(*
SPDX-FileCopyrightText: © 2026 Oleksandr Tiutyk <trofimich@gmail.com>
SPDX-License-Identifier: MIT
License: https://opensource.org/license/mit
*)

(*!
<summary>Stores unique generic values with fixed or dynamic capacity.</summary>
<description>
CreateEnumerator allocates an independent cursor owned by its caller. The collection must remain alive while
that cursor is used. SetGeneric replaces a matching entry with the incoming descriptor. SetGeneric preserves
disposal responsibility when the same allocation is reused; transferred caller-side owning aliases must not be
released again. Lookup uses GENERIC_VALUE equality/hashing or the borrowed valueEqualityComparer supplied once
through FB_init. Pass zero explicitly to use default value equality and hashing. Empty values are supported
unless rejected by a validator. Raw queries create borrowed descriptors with an explicit object flag. Entries
and enumeration have no guaranteed order; positions are storage slots, not sorted ranks. Do not modify stored
descriptors through returned references. Try lookup/removal operations contain exceptions without rolling back
partial effects. Generic query arguments are borrowed by default. Explicitly requested release in Try
operations is attempted even after lookup failure; caller-side owning aliases are not reset. Borrowed
elements, including OBJECT instances, remain caller-owned and must stay alive while stored. Do not delete
owned payload through external aliases. Keep equality/hash-relevant data and comparer configuration stable:
remove before changing them, then insert again. Fields unrelated to active equality/hash may change. Callbacks
must not mutate elements or reenter collection mutation; explicit query release must not dispose of retained
storage. Default OBJECT equality/hashing uses Object.Equals/GetHashCode; Clone has its own identity. Discard
and populate the index again after equality-relevant address relocation before further lookup. Static index
storage adds 12 bytes per capacity slot and three pointers plus the comparer reference. Dynamic entries and
the 12-byte-per-slot index share one allocation; growth temporarily retains both old and new allocations.
Expected bucket lookup is constant time plus hashing/equality costs, worst case linear; compaction and
rebuilding after removal are linear in capacity and Length. The validator is borrowed for the collection
lifetime. No internal locking is implemented. Concurrent access involving mutation requires caller
coordination; this implementation does not provide a concurrent-container guarantee. Generic lookup with
requested query release also attempts cleanup on lookup failure before propagating the captured exception;
terminal OOM takes precedence.
Instances cannot be assigned by value: copying backing pointers or disposal responsibility would create
unsafe aliases. Interface references still borrow this instance; copying an interface does not clone storage.
</description>
*)

{attribute 'no_explicit_call' := 'do not call this function block directly'}
FUNCTION_BLOCK UniqueDataSet
VAR_GENERIC CONSTANT
	{attribute 'hide'}
	//! <summary>Inline capacity; zero selects dynamic backing storage.</summary>
	_StaticCapacity : TOF_Core.DINT_LENGTH := 0;
END_VAR
EXTENDS TOF_Core.Object IMPLEMENTS IUniqueDataSet
VAR_INPUT
	//! <summary>Number of slots added when dynamic storage is full; must be positive when growth is required.</summary>
	DefaultDynamicAllocationElementCount : BYTE := 10;
END_VAR
VAR_STAT
	//! <summary>Class name shared by all instances of this function block.</summary>
	{attribute 'hide'}
	_ClassName : STRING := __POUNAME();
END_VAR
VAR
	{attribute 'hide'}
	_ValueValidator : TOF_Core.IGenericValueValidator;
	{attribute 'hide'}
	_ValueEqualityComparer : TOF_Core.IEqualityComparer;

	{attribute 'hide'}
	_Array : POINTER TO TOF_Core.GENERIC_VALUE;
	{attribute 'hide'}
	_StaticArray : ARRAY [0.._StaticCapacity - 1] OF TOF_Core.GENERIC_VALUE;

	{attribute 'hide'}
	_Hashes : POINTER TO UDINT;
	{attribute 'hide'}
	_Buckets : POINTER TO DINT;
	{attribute 'hide'}
	_NextIndices : POINTER TO DINT;

	{attribute 'hide'}
	_StaticHashes : ARRAY [0.._StaticCapacity - 1] OF UDINT;
	{attribute 'hide'}
	_StaticBuckets : ARRAY [0.._StaticCapacity - 1] OF DINT;
	{attribute 'hide'}
	_StaticNextIndices : ARRAY [0.._StaticCapacity - 1] OF DINT;

	{attribute 'hide'}
	_DynamicCapacity : TOF_Core.DINT_LENGTH;
	{attribute 'hide'}
	_Length : TOF_Core.DINT_LENGTH;
END_VAR

(*!
<summary>Grows the combined entry and hash-index buffer before accepting incoming ownership.</summary>
<description>
Static collections return without allocation. A positive increment must fit DINT capacity and the UDINT
allocation-byte limit, including 12 index bytes per slot. One allocation contains entries, cached hashes,
bucket heads and links. Allocation failure preserves the old buffer, index, capacity and payload ownership and
sets terminal allocation state. Existing descriptors and hashes are copied; rebuilding links invokes no
equality/hash callbacks. Descendants cannot override this storage operation; capacity, indexing and disposal
remain governed by this collection implementation.
</description>
*)
METHOD PROTECTED FINAL AllocateMemory
VAR_INPUT
	elementCount : TOF_Core.DINT_LENGTH;
END_VAR
VAR CONSTANT
	//! <summary>Bytes per capacity slot, including descriptor storage and any hash-index arrays.</summary>
	ENTRY_ALLOCATION_SIZE : ULINT := XSIZEOF(TOF_Core.GENERIC_VALUE) + XSIZEOF(UDINT) + 2 * XSIZEOF(DINT);
END_VAR
VAR
	newMemory : POINTER TO BYTE;
	newHashes : POINTER TO UDINT;
	newCapacity : ULINT;

END_VAR
IF NOT Dynamic THEN
	RETURN;
END_IF

IF elementCount <= TOF_Core.SignedInt32.ZERO THEN
	TOF_Core.Exceptions.ThrowArgumentOutOfRange(
		sourceNamespaceName := NamespaceName,
		sourceClassName := ClassName,
		sourcePOUName := __POUNAME(),
		sourcePosition := __POSITION(),
		argumentName := 'elementCount',
		argumentValue := elementCount
	);
END_IF

newCapacity := TO_ULINT(_DynamicCapacity) + TO_ULINT(elementCount);

IF newCapacity > TO_ULINT(TOF_Core.SignedInt32.MAX_VALUE)
	OR_ELSE newCapacity > TO_ULINT(TOF_Core.UnsignedInt32.MAX_VALUE) / ENTRY_ALLOCATION_SIZE
THEN
	TOF_Core.Exceptions.ThrowArgumentOutOfRange(
		sourceNamespaceName := NamespaceName,
		sourceClassName := ClassName,
		sourcePOUName := __POUNAME(),
		sourcePosition := __POSITION(),
		argumentName := 'capacity',
		argumentValue := newCapacity
	);
END_IF

newMemory := __NEW(BYTE, TO_UDINT(ENTRY_ALLOCATION_SIZE * newCapacity));

IF newMemory = 0 THEN
	TOF_Core.DynamicMemoryManager.RaiseAllocationFailure();
END_IF

newHashes := newMemory + TO_UDINT(XSIZEOF(TOF_Core.GENERIC_VALUE) * newCapacity);

IF _Length > TOF_Core.SignedInt32.ZERO THEN
	Tc2_System.MEMCPY(
		destAddr := newMemory,
		srcAddr := _Array,
		n := TO_UDINT(XSIZEOF(TOF_Core.GENERIC_VALUE) * TO_ULINT(_Length))
	);
	Tc2_System.MEMCPY(destAddr := newHashes, srcAddr := _Hashes, n := TO_UDINT(XSIZEOF(UDINT) * TO_ULINT(_Length)));
END_IF

IF _Array <> 0 THEN
	__DELETE(_Array);
END_IF

_Array := newMemory;
_Hashes := newHashes;
_Buckets := newMemory + TO_UDINT((XSIZEOF(TOF_Core.GENERIC_VALUE) + XSIZEOF(UDINT)) * newCapacity);
_NextIndices := newMemory + TO_UDINT((XSIZEOF(TOF_Core.GENERIC_VALUE) + XSIZEOF(UDINT) + XSIZEOF(DINT)) * newCapacity);
_DynamicCapacity := TO_DINT(newCapacity);

rebuildIndex();
END_METHOD

(*!
<summary>Reports the currently allocated number of slots.</summary>
<description>
Units are bytes for ByteList and entries for other collections. Static capacity is fixed; dynamic capacity can
change on growth or clearing. This is not a guarantee that the next allocation succeeds.
</description>
*)
{attribute 'monitoring' := 'call'}
PROPERTY FINAL Capacity : TOF_Core.DINT_LENGTH
GET
Capacity := SEL(_StaticCapacity = 0, _StaticCapacity, _DynamicCapacity);
END_GET
END_PROPERTY

(*!
<summary>Borrows the concrete collection class name without transferring storage ownership.</summary>
*)
{attribute 'monitoring' := 'call'}
PROPERTY ClassName : REFERENCE TO STRING
GET
ClassName REF= _ClassName;
END_GET
END_PROPERTY

(*!
<summary>Removes all entries and releases dynamic entry and index storage.</summary>
<description>
Owned payload cleanup is best effort. The collection is marked empty before disposal; cleanup callbacks must
not reenter mutation. Static capacity and the lifetime comparer/validators are retained. Dynamic capacity
becomes zero. Uses no allocation or equality/hash callbacks and leaves static buckets empty for reuse.
Descendants cannot override this storage operation; capacity, indexing and disposal remain governed by this
collection implementation.
</description>
*)
METHOD FINAL Clear : IUniqueDataSet
VAR
	index : DINT;
	entryCount : DINT;
END_VAR
Clear := THIS^;
entryCount := _Length;
_Length := 0;

FOR index := 0 TO entryCount - 1 DO
	_Array[index].Release();
END_FOR

IF Dynamic THEN
	IF _Array <> 0 THEN
		__DELETE(_Array);
	END_IF

	_Array := 0;
	_Hashes := 0;
	_Buckets := 0;
	_NextIndices := 0;
	_DynamicCapacity := 0;
ELSE
	rebuildIndex();
END_IF
END_METHOD

(*!
<summary>Reports whether a matching raw query exists.</summary>
<description>
The raw ANY argument is borrowed without cloning or ownership transfer. isObject = TRUE requires a live Object
function-block instance, not a pointer or interface variable. FALSE uses ordinary runtime type mapping. The
caller keeps the query storage alive for the call. Descendants cannot override this storage operation;
capacity, indexing and disposal remain governed by this collection implementation.
</description>
*)
//!<param name="isObject">Explicitly interprets the raw argument as a live Object instance.</param>
METHOD FINAL Contains : BOOL
VAR_INPUT
	value : ANY;
	isObject : BOOL := FALSE;
END_VAR
VAR
	genericValue : TOF_Core.GENERIC_VALUE;
END_VAR

genericValue := TOF_Core.GenericValueFactory.FromAnyType(
		value := value,
		isObject := isObject,
		memoryManagementBehavior := TOF_Core.GENERIC_MEMORY_MANAGEMENT_BEHAVIOR.STORE_ORIGINAL_REFERENCE_AND_NOT_OWNS_MEMORY
	);

Contains := FindIndex(value := genericValue);
END_METHOD

(*!
<summary>Reports whether a matching entry exists for a borrowed generic query.</summary>
<description>
The query is borrowed by default. Explicit release requests disposal of owned query storage after lookup
completes, including a missing result. Requested release is attempted after both successful lookup and lookup
failure. Before cleanup, the original framework exception is retained and a borrowed static system exception
is cloned to preserve its code, catch point and timestamps across cleanup callbacks. The captured exception is
then propagated through ExceptionManager.Throw in the current cyclic task; native errors use the framework
SystemException representation. If capturing the system exception fails with terminal OOM, query cleanup is
still attempted and terminal OOM takes precedence. Terminal allocation state is never cleared. Release is best
effort and does not prove successful deallocation. Cleanup callbacks must not reenter collection mutation.
Release resets only the local descriptor copy; the caller must have disposal rights and must not reuse or
release owning aliases afterwards. Borrowed payload is not freed. Descendants cannot override this storage
operation; capacity, indexing and disposal remain governed by this collection implementation.
</description>
*)
METHOD FINAL ContainsGeneric : BOOL
VAR_INPUT
	value : TOF_Core.GENERIC_VALUE;
	releaseValue : BOOL := FALSE;
END_VAR
VAR
	exceptionCode : __SYSTEM.ExceptionCode;
	caughtException : TOF_Core.IException;
END_VAR
__TRY
	ContainsGeneric := FindIndex(value := value);
__CATCH(exceptionCode)
	caughtException := TOF_Core.ExceptionManager.GetLastException(
		exceptionCode := exceptionCode,
		catchPointNamespaceName := NamespaceName,
		catchPointPOUName := __POUNAME(),
		catchPointPosition := __POSITION()
	);
__ENDTRY

IF releaseValue THEN
	IF caughtException <> 0 AND_THEN NOT caughtException.IsDynamicInstance THEN
		__TRY
			TOF_Core.DynamicMemoryManager.RaiseIfAllocationFailed();
			__QUERYINTERFACE(caughtException.Clone(), caughtException);
		__CATCH(exceptionCode)
			value.Release();

			TOF_Core.ExceptionManager.ReThrowLastException(
				exceptionCode := exceptionCode,
				catchPointNamespaceName := NamespaceName,
				catchPointPOUName := __POUNAME(),
				catchPointPosition := __POSITION()
			);
		__ENDTRY
	END_IF

	value.Release();
END_IF

IF caughtException <> 0 THEN
	TOF_Core.ExceptionManager.Throw(exception := caughtException);
END_IF
END_METHOD

(*!
<summary>Creates an independent enumerator owned by the caller.</summary>
<description>
The caller must explicitly release the enumerator and keep this collection alive while using it. Allocation
failure invokes DynamicMemoryManager.RaiseAllocationFailure without a heap exception; it is terminal and is
not returned as a recoverable null result.
</description>
*)
METHOD CreateEnumerator : TOF_Core.IEnumerator
VAR
	enumerator : POINTER TO UniqueDataSetEnumerator;
END_VAR
enumerator := __NEW(UniqueDataSetEnumerator(uniqueSet := THIS^));

IF enumerator = 0 THEN
	TOF_Core.DynamicMemoryManager.RaiseAllocationFailure();
END_IF

CreateEnumerator := enumerator^;
END_METHOD

(*!
<summary>Reports whether storage can grow dynamically.</summary>
<description>
Static capacity zero selects dynamic storage. Dynamic collections can still fail to allocate.
</description>
*)
{attribute 'monitoring' := 'call'}
PROPERTY FINAL Dynamic : BOOL
GET
Dynamic := _StaticCapacity = 0;
END_GET
END_PROPERTY

(*!
<summary>Reports whether the collection has no entries.</summary>
<description>
Reflects Length; not a check of payload lifetime or memory health.
</description>
*)
{attribute 'monitoring' := 'call'}
PROPERTY FINAL Empty : BOOL
GET
Empty := _Length <= 0;
END_GET
END_PROPERTY

(*!
<summary>Releases collection payload and dynamic entry/index storage during destruction.</summary>
<description>
Calls the non-allocating Clear path without invoking equality/hash callbacks. Owned payload release is best
effort and cannot guarantee successful deallocation; cleanup callbacks must not throw or reenter mutation.
</description>
*)

METHOD FB_exit : BOOL
VAR_INPUT
	bInCopyCode : BOOL;
END_VAR
Clear();
END_METHOD

(*!
<summary>Binds the validator, the lifetime equality strategy and static storage.</summary>
<description>
The value comparer is borrowed for the entire collection lifetime. Supply it explicitly; zero selects
GENERIC_VALUE default equality and hashing. Keep it alive and its equality-relevant configuration stable.
There is no subsequent comparer replacement. Initialization binds existing storage without allocating or
calling validators, comparers or other throwing paths.
</description>
*)


//!<param name="valueEqualityComparer">
//! Borrowed value equality and hash strategy; pass zero explicitly for the GENERIC_VALUE defaults.
//! </param>
METHOD FB_init : BOOL
VAR_INPUT
	bInitRetains : BOOL; // TRUE: the retain variables are initialized (reset warm / reset cold)
	bInCopyCode : BOOL; // TRUE: the instance will be copied to the copy code afterward (online change)

	valueValidator : TOF_Core.IGenericValueValidator;
	valueEqualityComparer : TOF_Core.IEqualityComparer;
END_VAR
_ValueValidator := valueValidator;
_ValueEqualityComparer := valueEqualityComparer;

IF NOT Dynamic THEN
	_Array := ADR(_StaticArray);
	_Hashes := ADR(_StaticHashes);
	_Buckets := ADR(_StaticBuckets);
	_NextIndices := ADR(_StaticNextIndices);
END_IF
END_METHOD

(*!
<summary>Finds an equal value through its hash bucket.</summary>
<description>
Borrows the descriptor and payload without changing ownership. The configured equality strategy computes the
query hash once; equal hash codes are resolved with Equals. Callback exceptions propagate before mutation. On
a miss supposedIndex is the append position. hashCode is valid after a completed lookup, including a miss. No
ordering or sorted rank is provided. Bucket heads and links encode entry index plus one; zero ends a chain.
Descendants cannot override this storage operation; capacity, indexing and disposal remain governed by this
collection implementation.
</description>
*)
METHOD PROTECTED FINAL FindIndex : BOOL
VAR_INPUT
	value : TOF_Core.GENERIC_VALUE;
END_VAR
VAR_OUTPUT
	supposedIndex : DINT;
	hashCode : UDINT;
END_VAR
VAR
	entryLink : DINT;
	entryIndex : DINT;
END_VAR
FindIndex := FALSE;
supposedIndex := _Length;
hashCode := value.GetHashCode(comparer := _ValueEqualityComparer);

IF _Length = TOF_Core.SignedInt32.ZERO THEN
	RETURN;
END_IF

entryLink := _Buckets[TO_DINT(hashCode MOD TO_UDINT(Capacity))];

WHILE entryLink <> TOF_Core.SignedInt32.ZERO DO
	entryIndex := entryLink - 1;

	IF _Hashes[entryIndex] = hashCode
		AND_THEN _Array[entryIndex].Equals(otherValue := value, comparer := _ValueEqualityComparer)
	THEN
		supposedIndex := entryIndex;
		FindIndex := TRUE;
		RETURN;
	END_IF

	entryLink := _NextIndices[entryIndex];
END_WHILE
END_METHOD

(*!
<summary>Reports whether fixed-capacity storage has no free slot.</summary>
<description>
Dynamic collections report FALSE even when Length equals Capacity. This does not guarantee available heap
memory.
</description>
*)
{attribute 'monitoring' := 'call'}
PROPERTY FINAL Full : BOOL
GET
Full := _StaticCapacity <> 0 AND_THEN _Length >= _StaticCapacity;
END_GET
END_PROPERTY

(*!
<summary>Borrows the entry at a current storage position.</summary>
<description>
The index must be within Length and is not a sorted rank; otherwise an exception is raised. The returned
descriptor reference and payload remain collection-owned or borrowed from their original owner. Do not mutate
the descriptor or dispose of its payload through this view. Mutation or destruction may invalidate the
reference. Descendants cannot override this storage operation; capacity, indexing and disposal remain governed
by this collection implementation.
</description>
*)
METHOD FINAL GetByIndex : REFERENCE TO TOF_Core.GENERIC_VALUE
VAR_INPUT
	index : DINT;
END_VAR
IF index < 0 OR_ELSE index >= _Length THEN
	TOF_Core.Exceptions.ThrowArgumentOutOfRange(
		sourceNamespaceName := NamespaceName,
		sourceClassName := ClassName,
		sourcePOUName := __POUNAME(),
		sourcePosition := __POSITION(),
		argumentName := 'index',
		argumentValue := index
	);
END_IF

GetByIndex REF= _Array[index];
END_METHOD

(*!
<summary>Returns the matching entry position, or a negative value when absent.</summary>
<description>
The query is borrowed by default. Explicit release requests disposal of owned query storage after lookup
completes, including a missing result. Requested release is attempted after both successful lookup and lookup
failure. Before cleanup, the original framework exception is retained and a borrowed static system exception
is cloned to preserve its code, catch point and timestamps across cleanup callbacks. The captured exception is
then propagated through ExceptionManager.Throw in the current cyclic task; native errors use the framework
SystemException representation. If capturing the system exception fails with terminal OOM, query cleanup is
still attempted and terminal OOM takes precedence. Terminal allocation state is never cleared. Release is best
effort and does not prove successful deallocation. Cleanup callbacks must not reenter collection mutation.
Release resets only the local descriptor copy; the caller must have disposal rights and must not reuse or
release owning aliases afterwards. Borrowed payload is not freed. The position is a current storage slot with
no sorted-rank guarantee; mutation may invalidate it. Descendants cannot override this storage operation;
capacity, indexing and disposal remain governed by this collection implementation.
</description>
*)
METHOD FINAL GetGenericValuePosition : DINT
VAR_INPUT
	value : TOF_Core.GENERIC_VALUE;
	releaseValue : BOOL := FALSE;
END_VAR
VAR
	exceptionCode : __SYSTEM.ExceptionCode;
	caughtException : TOF_Core.IException;
END_VAR
__TRY
	IF NOT FindIndex(value := value, supposedIndex => GetGenericValuePosition) THEN
		GetGenericValuePosition := -1;
	END_IF
__CATCH(exceptionCode)
	caughtException := TOF_Core.ExceptionManager.GetLastException(
		exceptionCode := exceptionCode,
		catchPointNamespaceName := NamespaceName,
		catchPointPOUName := __POUNAME(),
		catchPointPosition := __POSITION()
	);
__ENDTRY

IF releaseValue THEN
	IF caughtException <> 0 AND_THEN NOT caughtException.IsDynamicInstance THEN
		__TRY
			TOF_Core.DynamicMemoryManager.RaiseIfAllocationFailed();
			__QUERYINTERFACE(caughtException.Clone(), caughtException);
		__CATCH(exceptionCode)
			value.Release();

			TOF_Core.ExceptionManager.ReThrowLastException(
				exceptionCode := exceptionCode,
				catchPointNamespaceName := NamespaceName,
				catchPointPOUName := __POUNAME(),
				catchPointPosition := __POSITION()
			);
		__ENDTRY
	END_IF

	value.Release();
END_IF

IF caughtException <> 0 THEN
	TOF_Core.ExceptionManager.Throw(exception := caughtException);
END_IF
END_METHOD

(*!
<summary>Returns the matching storage position, or a negative value when absent.</summary>
<description>
The raw ANY argument is borrowed without cloning or ownership transfer. isObject = TRUE requires a live Object
function-block instance, not a pointer or interface variable. FALSE uses ordinary runtime type mapping. The
caller keeps the query storage alive for the call. The position is a current storage slot with no sorted-rank
guarantee; mutation may invalidate it. Descendants cannot override this storage operation; capacity, indexing
and disposal remain governed by this collection implementation.
</description>
*)
//!<param name="isObject">Explicitly interprets the raw argument as a live Object instance.</param>
METHOD FINAL GetValuePosition : DINT
VAR_INPUT
	value : ANY;
	isObject : BOOL := FALSE;
END_VAR
VAR
	genericValue : TOF_Core.GENERIC_VALUE;
END_VAR

genericValue := TOF_Core.GenericValueFactory.FromAnyType(
		value := value,
		isObject := isObject,
		memoryManagementBehavior := TOF_Core.GENERIC_MEMORY_MANAGEMENT_BEHAVIOR.STORE_ORIGINAL_REFERENCE_AND_NOT_OWNS_MEMORY
	);

IF NOT FindIndex(value := genericValue, supposedIndex => GetValuePosition) THEN
	GetValuePosition := -1;
END_IF
END_METHOD

(*!
<summary>Reports the number of stored entries.</summary>
<description>
Units are bytes for ByteList and entries for other collections. Existing positions range from zero through
Length minus one.
</description>
*)
{attribute 'monitoring' := 'call'}
PROPERTY FINAL Length : TOF_Core.DINT_LENGTH
GET
Length := _Length;
END_GET
END_PROPERTY

(*!
<summary>Provides the library namespace for diagnostics.</summary>
<description>
Borrowed read-only reference to compiler-initialized metadata; no ownership transfer.
</description>
*)
{attribute 'monitoring' := 'call'}
PROPERTY NamespaceName : REFERENCE TO STRING
GET
NamespaceName REF= CurrentNamespace.Name;
END_GET
END_PROPERTY

(*!
<summary>Rebuilds bucket chains from cached hashes after entry relocation or capacity changes.</summary>
<description>
Requires bound index storage for positive capacity and valid hashes for every live entry. Does not allocate,
access payload or invoke callbacks. This only rebuilds links; it does not recompute hashes after
equality-relevant payload or address changes.
</description>
*)
METHOD PRIVATE rebuildIndex
VAR
	index : DINT;
	bucketIndex : DINT;
END_VAR
IF Capacity = TOF_Core.SignedInt32.ZERO THEN
	RETURN;
END_IF

Tc2_System.MEMSET(destAddr := _Buckets, fillByte := 0, n := TO_UDINT(XSIZEOF(DINT) * TO_ULINT(Capacity)));

FOR index := 0 TO _Length - 1 DO
	bucketIndex := TO_DINT(_Hashes[index] MOD TO_UDINT(Capacity));
	_NextIndices[index] := _Buckets[bucketIndex];
	_Buckets[bucketIndex] := index + 1;
END_FOR
END_METHOD

(*!
<summary>Removes the entry at a current storage position.</summary>
<description>
The index must be within Length and is not a sorted rank. Entries after the removed slot are compacted and
bucket links rebuilt from cached hashes before owned payload cleanup. Index compaction and rebuilding invoke
no equality/hash callbacks and allocate no storage. Invalid indices raise an exception. Positions and borrowed
entry references may be invalidated. Payload disposal is best effort through GENERIC_VALUE.Release.
Descendants cannot override this storage operation; capacity, indexing and disposal remain governed by this
collection implementation.
</description>
*)
METHOD FINAL RemoveAt : IUniqueDataSet
VAR_INPUT
	index : DINT;
END_VAR
VAR
	removedValue : TOF_Core.GENERIC_VALUE;
END_VAR
IF index < TOF_Core.SignedInt32.ZERO OR_ELSE index >= _Length THEN
	TOF_Core.Exceptions.ThrowArgumentOutOfRange(
		sourceNamespaceName := NamespaceName,
		sourceClassName := ClassName,
		sourcePOUName := __POUNAME(),
		sourcePosition := __POSITION(),
		argumentName := 'index',
		argumentValue := index
	);
END_IF

RemoveAt := THIS^;
removedValue := _Array[index];

IF index < _Length - 1 THEN
	Tc2_System.MEMMOVE(
		destAddr := ADR(_Array[index]),
		srcAddr := ADR(_Array[index + 1]),
		n := TO_UDINT(XSIZEOF(TOF_Core.GENERIC_VALUE) * TO_ULINT(_Length - index - 1))
	);
	Tc2_System.MEMMOVE(
		destAddr := ADR(_Hashes[index]),
		srcAddr := ADR(_Hashes[index + 1]),
		n := TO_UDINT(XSIZEOF(UDINT) * TO_ULINT(_Length - index - 1))
	);
END_IF

_Array[_Length - 1].Reset();
_Length := _Length - 1;
rebuildIndex();

removedValue.Release();
END_METHOD

(*!
<summary>Reports the size of this function-block instance.</summary>
<description>
Measured in bytes; includes inline storage but excludes separately allocated buffers, payload and enumerators.
</description>
*)
{attribute 'monitoring' := 'call'}
PROPERTY SelfSize : ULINT
GET
SelfSize := XSIZEOF(THIS^);
END_GET
END_PROPERTY

(*!
<summary>Copies a value and stores it through SetGeneric.</summary>
<description>
Borrows the original during the call. isObject = TRUE requires a live Object FB instance implementing
ICloneable; other data is copied as bytes without recursively cloning references. A prepared copy is released
if insertion fails before acceptance; exceptions propagate. Engine-managed exception objects are unsupported.
Any index output is meaningful only on success. Descendants cannot override this storage operation; capacity,
indexing and disposal remain governed by this collection implementation.
The original failure is captured before cleanup so nested cleanup handling cannot replace its payload.
A static native wrapper is cloned before cleanup; failure to capture still attempts prepared-copy disposal.
Terminal allocation failure takes precedence and no exception clone is allocated after its latch is set.
</description>
*)
METHOD FINAL SetCopy : IUniqueDataSet
VAR_INPUT
	value : ANY;
	isObject : BOOL := FALSE;
END_VAR
VAR_OUTPUT
	index : DINT;
END_VAR
VAR
	exceptionCode : __SYSTEM.ExceptionCode;
	caughtException : TOF_Core.IException;
	genericValue : TOF_Core.GENERIC_VALUE;
END_VAR

genericValue := TOF_Core.GenericValueFactory.FromAnyType(
		value := value,
		isObject := isObject,
		memoryManagementBehavior := TOF_Core.GENERIC_MEMORY_MANAGEMENT_BEHAVIOR.CLONE_ORIGINAL_VALUE_AND_OWNS_MEMORY
	);

__TRY
	SetCopy := SetGeneric(value := genericValue, index => index);
__CATCH(exceptionCode)
	caughtException := TOF_Core.ExceptionManager.GetLastException(
		exceptionCode := exceptionCode,
		catchPointNamespaceName := NamespaceName,
		catchPointPOUName := __POUNAME(),
		catchPointPosition := __POSITION()
	);
__ENDTRY

IF caughtException <> 0 THEN
	__TRY
		TOF_Core.DynamicMemoryManager.RaiseIfAllocationFailed();

		IF NOT caughtException.IsDynamicInstance THEN
			__QUERYINTERFACE(caughtException.Clone(), caughtException);
		END_IF
	__CATCH(exceptionCode)
		genericValue.Release();

		TOF_Core.ExceptionManager.ReThrowLastException(
			exceptionCode := exceptionCode,
			catchPointNamespaceName := NamespaceName,
			catchPointPOUName := __POUNAME(),
			catchPointPosition := __POSITION()
		);
	__ENDTRY

	genericValue.Release();

	TOF_Core.ExceptionManager.Throw(exception := caughtException);
END_IF
END_METHOD

(*!
<summary>Inserts a value or replaces the matching entry with the incoming descriptor.</summary>
<description>
Uses the lifetime equality/hash strategy, with no ordering guarantee. Empty descriptors are permitted unless
rejected by a validator. A successful call accepts incoming owned storage; borrowed payload must remain alive
while stored. Validation, lookup and growth precede acceptance; failure before acceptance leaves ownership
with the caller. A displaced owned allocation is released after replacement. Reusing the same allocation does
not release it and preserves existing ownership or accepts incoming ownership, without implicitly returning
ownership to the caller. Caller-side descriptor copies are not reset; transferred owning aliases must not be
released or reused as owners. Aliases must have compatible disposal semantics; overlapping owned ranges and
ownership already held by another entry or owner are not supported. Callbacks must not mutate or reenter this
collection. Cleanup through GENERIC_VALUE.Release is best effort and does not guarantee deallocation. The
index output is valid only on success. Descendants cannot override this storage operation; capacity, indexing
and disposal remain governed by this collection implementation.
</description>
*)
//!<param name="value">Incoming descriptor; owned storage is transferred on success.</param>
METHOD FINAL SetGeneric : IUniqueDataSet
VAR_INPUT
	value : TOF_Core.GENERIC_VALUE;
END_VAR
VAR_OUTPUT
	index : DINT;
END_VAR
VAR

	supposedIndex : DINT;
	hashCode : UDINT;
	bucketIndex : DINT;

	displacedValue : TOF_Core.GENERIC_VALUE;
END_VAR
IF _ValueValidator <> 0 THEN
	_ValueValidator.Validate(validatedObjectName := GetName(), valueToValidate := value);
END_IF

SetGeneric := THIS^;

IF FindIndex(value := value, supposedIndex => supposedIndex, hashCode => hashCode) THEN
	displacedValue := _Array[supposedIndex];

	IF displacedValue.Address = value.Address THEN
		IF displacedValue.IsMemoryOwner AND_THEN NOT value.IsMemoryOwner THEN
			value := TOF_Core.GenericValueFactory.FromParts(
				genericTypeClass := value.TypeClass,
				address := value.Address,
				size := value.Size,
				memoryManagementBehavior := TOF_Core.GENERIC_MEMORY_MANAGEMENT_BEHAVIOR.STORE_ORIGINAL_REFERENCE_AND_OWNS_MEMORY
			);
		END_IF

		displacedValue.Reset();
	END_IF
ELSE
	IF _Length >= Capacity THEN
		IF Dynamic THEN
			AllocateMemory(elementCount := DefaultDynamicAllocationElementCount);
		ELSE
			TOF_Core.Exceptions.ThrowStaticCollectionFull(
				sourceNamespaceName := NamespaceName,
				sourceClassName := ClassName,
				sourcePOUName := __POUNAME(),
				sourcePosition := __POSITION(),
				collectionName := GetName(),
				capacity := TO_UDINT(Capacity)
			);
		END_IF
	END_IF
END_IF

_Array[supposedIndex] := value;

IF supposedIndex = _Length THEN
	_Hashes[supposedIndex] := hashCode;
	bucketIndex := TO_DINT(hashCode MOD TO_UDINT(Capacity));
	_NextIndices[supposedIndex] := _Buckets[bucketIndex];
	_Buckets[bucketIndex] := supposedIndex + 1;
	_Length := _Length + 1;
END_IF

displacedValue.Release();

index := supposedIndex;
END_METHOD

(*!
<summary>Attempts to remove a matching entry.</summary>
<description>
Returns the collection for chaining. removed is TRUE only after the matching entry has been removed; FALSE
means no completed removal was reported. Removal is not transactional and does not prove successful
destruction of an owned payload. Catches exceptions without propagating them or clearing terminal allocation
state. Partial changes are not rolled back. The raw ANY argument is borrowed without cloning or ownership
transfer. isObject = TRUE requires a live Object function-block instance, not a pointer or interface variable.
FALSE uses ordinary runtime type mapping. The caller keeps the query storage alive for the call. Descendants
cannot override this storage operation; capacity, indexing and disposal remain governed by this collection
implementation.
After nested calls and requested cleanup, a fatal allocation state forces the reported outcome to failure.
This does not roll back completed removal or reset the application-wide fatal latch.
</description>
*)
//!<param name="isObject">Explicitly interprets the raw argument as a live Object instance.</param>
METHOD FINAL TryRemove : IUniqueDataSet
VAR_INPUT
	value : ANY;
	isObject : BOOL := FALSE;
END_VAR
VAR_OUTPUT
	removed : BOOL;
END_VAR
VAR
	genericValue : TOF_Core.GENERIC_VALUE;
	index : DINT;
END_VAR
TryRemove := THIS^;
removed := FALSE;

__TRY
	genericValue := TOF_Core.GenericValueFactory.FromAnyType(
		value := value,
		isObject := isObject,
		memoryManagementBehavior := TOF_Core.GENERIC_MEMORY_MANAGEMENT_BEHAVIOR.STORE_ORIGINAL_REFERENCE_AND_NOT_OWNS_MEMORY
	);

	IF FindIndex(value := genericValue, supposedIndex => index) THEN
		RemoveAt(index := index);
		removed := TRUE;
	END_IF
__CATCH
	removed := FALSE;
__ENDTRY

IF TOF_Core.DynamicMemoryManager.HasAllocationFailed THEN
	removed := FALSE;
END_IF
END_METHOD

(*!
<summary>Attempts to remove a matching entry.</summary>
<description>
Returns the collection for chaining. removed is TRUE only after the matching entry has been removed; FALSE
means no completed removal was reported. Removal is not transactional and does not prove successful
destruction of an owned payload. Catches exceptions without propagating them or clearing terminal allocation
state. Partial changes are not rolled back. The query is borrowed by default. When releaseValue is explicitly
TRUE, attempts to release the supplied generic argument after lookup/removal even on failure. The caller must
have disposal rights and must not reuse aliases of an owned argument after release. Descendants cannot
override this storage operation; capacity, indexing and disposal remain governed by this collection
implementation.
After nested calls and requested cleanup, a fatal allocation state forces the reported outcome to failure.
This does not roll back completed removal or reset the application-wide fatal latch.
</description>
*)
METHOD FINAL TryRemoveGeneric : IUniqueDataSet
VAR_INPUT
	value : TOF_Core.GENERIC_VALUE;
	releaseValue : BOOL := FALSE;
END_VAR
VAR_OUTPUT
	removed : BOOL;
END_VAR
VAR
	index : DINT;
END_VAR
TryRemoveGeneric := THIS^;
removed := FALSE;

__TRY
	IF FindIndex(value := value, supposedIndex => index) THEN
		RemoveAt(index := index);
		removed := TRUE;
	END_IF
__CATCH
	removed := FALSE;
__ENDTRY

IF releaseValue THEN
	__TRY
		value.Release();
	__CATCH
		removed := FALSE;
	__ENDTRY
END_IF

IF TOF_Core.DynamicMemoryManager.HasAllocationFailed THEN
	removed := FALSE;
END_IF
END_METHOD

(*!
<summary>Exposes the configured value validator.</summary>
<description>
Borrowed optional reference fixed at initialization. Zero means no validator. The collection does not own or
release it.
</description>
*)
{attribute 'monitoring' := 'call'}
PROPERTY FINAL ValueValidator : TOF_Core.IGenericValueValidator
GET
ValueValidator := _ValueValidator;
END_GET
END_PROPERTY

END_FUNCTION_BLOCK

(* stored: Version 1.1.0.1
   POU UniqueDataSet: Id {2442738f-11d0-404d-bb8d-7d07fa17599f}, SpecialFunc None
   Folder Service members: Id {ccb8ef2f-d434-4cac-96b9-34498b70bbbb}
   Method AllocateMemory: Id {27706325-8810-4759-a969-4aa4266a091f}
   Property Capacity: Id {442fc8a6-b0bb-403e-8549-1172e75c9349}
   Get Get: Id {9eba9911-6110-4fbb-bdf5-06f64345afad}
   Property ClassName: Id {467d00f1-7abe-4a3f-b6cd-fe49b224e254}
   Get Get: Id {252ee1d7-9d51-4251-a289-595ab545aa2e}
   Method Clear: Id {0def1be0-078f-4e42-b9d9-bacd7c63976c}
   Method Contains: Id {12fa0823-e803-4d25-984b-09daa27cbbd8}
   Method ContainsGeneric: Id {585b7317-248d-43d5-8f74-88f36cb9db8d}
   Method CreateEnumerator: Id {99cd46dc-a609-4207-b9f8-817b6841cc34}
   Property Dynamic: Id {4f4e7964-b376-49d8-b378-e30233cbcf40}
   Get Get: Id {74b076d1-9110-4644-a20a-753364c2a614}
   Property Empty: Id {43555ed7-74ac-45b4-80a6-0e3605f3c997}
   Get Get: Id {226fbd91-6757-4cc9-b8a9-dbade8a27ab4}
   Method FB_exit: Id {eb4ef8ca-4abf-497c-8a84-8766a913017b}
   Method FB_init: Id {e1f857c5-3b42-4120-8d16-dbd9cbb01e62}
   Method FindIndex: Id {24320c3b-fc49-4954-a0eb-fa84e7ceb897}
   Property Full: Id {c3e7f9e9-491d-47ed-b5be-e34cce8561b4}
   Get Get: Id {e784852e-9eaa-4e44-9445-b45c6bf3983e}
   Method GetByIndex: Id {8e83c179-a293-412f-8b67-0e71bf720692}
   Method GetGenericValuePosition: Id {080ff3a3-127e-451a-8f0f-949daec3002e}
   Method GetValuePosition: Id {d91713d1-b8ba-41d0-9834-7fd09ea4504a}
   Property Length: Id {9f5d9338-6134-422e-8cd0-945d2d30e1f6}
   Get Get: Id {d61178d6-0b1b-4e5d-a64d-f11834124588}
   Property NamespaceName: Id {e508ab9e-2295-4c2b-a61b-fa08b582c6ff}
   Get Get: Id {f6e5f586-787d-47e0-877c-e0fccdebc010}
   Method rebuildIndex: Id {780840c7-2bff-4fd3-b769-ff107364e1db}
   Method RemoveAt: Id {560da408-7178-47ba-9120-b01c5ed8fd70}
   Property SelfSize: Id {01bbb837-39f2-4ff6-93e9-d2a4ae7f8d4e}
   Get Get: Id {19f2cabd-ffd0-448b-9120-3e4def7ce2d6}
   Method SetCopy: Id {942d6884-b40d-46d4-872b-4443fcd5acea}
   Method SetGeneric: Id {e49ee7f0-ea9d-45ea-8ca1-9435721d8384}
   Method TryRemove: Id {83ed7c56-c31f-46ae-9dc0-2c64a9afa913}
   Method TryRemoveGeneric: Id {509dc21b-c80c-4a35-ad86-96721cdf54e6}
   Property ValueValidator: Id {0eab78c2-de3c-427a-9017-e6bb7fd4a1e3}
   Get Get: Id {0626a256-23ca-4414-bd79-e7c4da25d1dd} *)
